// LS Electric XG5000 project: 루시드 Test
// PLC NewPLC
// module base 0 slot 0: 입출력 모듈:XBM-DN32H (DC 24V입력/TR 출력, 32점)

PROGRAM NewProgram (task: 스캔 프로그램)

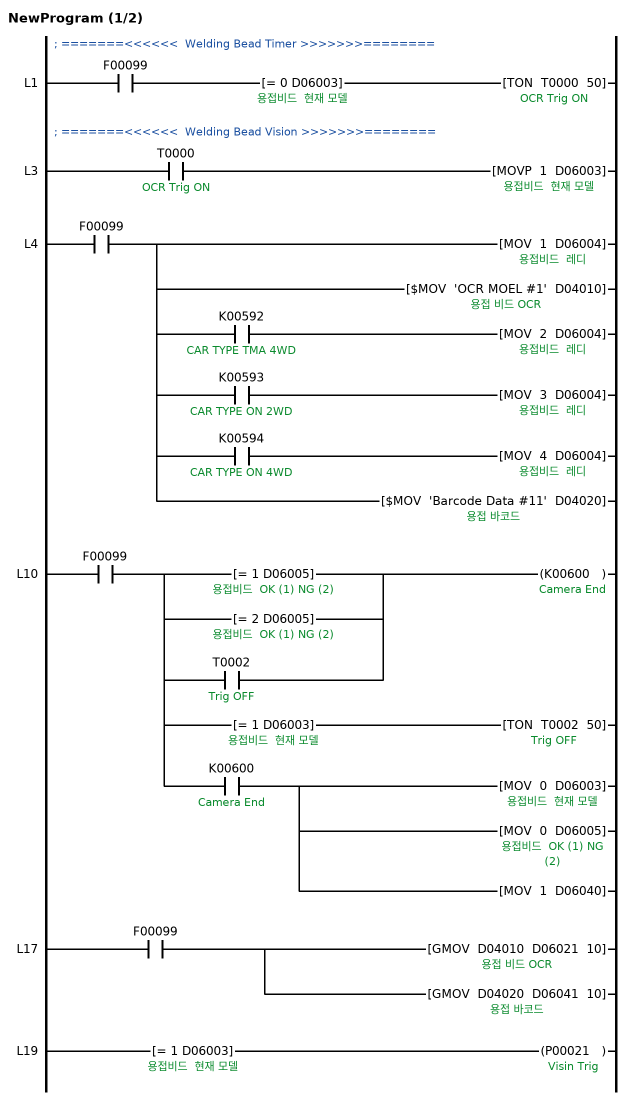
// =======<<<<<<  Welding Bead Timer >>>>>>>========
; L1
LOAD      F00099
AND=      0 D06003	// 용접비드  현재 모델
TON       T0000 50	// OCR Trig ON
// =======<<<<<<  Welding Bead Vision >>>>>>>========
; L3
LOAD      T0000	// OCR Trig ON
MOVP      1 D06003	// 용접비드  현재 모델
; L4
LOAD      F00099
MOV       1 D06004	// 용접비드  레디 
$MOV      'OCR MOEL #1' D04010	// 용접 비드 OCR
MPUSH
AND       K00592	// CAR TYPE TMA 4WD
MOV       2 D06004	// 용접비드  레디 
MLOAD
AND       K00593	// CAR TYPE ON 2WD
MOV       3 D06004	// 용접비드  레디 
MLOAD
AND       K00594	// CAR TYPE ON 4WD
MOV       4 D06004	// 용접비드  레디 
MPOP
$MOV      'Barcode Data #11' D04020	// 용접 바코드
; L10
LOAD      F00099
MPUSH
LOAD=     1 D06005	// 용접비드  OK (1) NG (2)
OR=       2 D06005	// 용접비드  OK (1) NG (2)
OR        T0002	// Trig OFF
AND LOAD
OUT       K00600	// Camera End
MLOAD
AND=      1 D06003	// 용접비드  현재 모델
TON       T0002 50	// Trig OFF
MPOP
AND       K00600	// Camera End
MOV       0 D06003	// 용접비드  현재 모델
MOV       0 D06005	// 용접비드  OK (1) NG (2)
MOV       1 D06040
; L17
LOAD      F00099
GMOV      D04010 D06021 10	// 용접 비드 OCR
GMOV      D04020 D06041 10	// 용접 바코드
; L19
LOAD=     1 D06003	// 용접비드  현재 모델
OUT       P00021	// Visin Trig

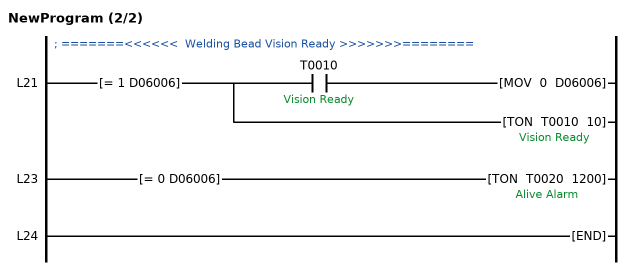
// =======<<<<<<  Welding Bead Vision Ready >>>>>>>========
; L21
LOAD=     1 D06006
MPUSH
AND       T0010	// Vision Ready
MOV       0 D06006
MPOP
TON       T0010 10	// Vision Ready
; L23
LOAD=     0 D06006
TON       T0020 1200	// Alive Alarm
; L24
END

VARIABLES AND COMMENTS (devices not used above)
D06000	WORD	용접비드  촬영 (1: 전송 0:PC)
D06001	WORD	용접비드  OCR 전송
D06002	WORD	용접비드  바코드 전송
K00591	BIT	CAR TYPE TMA 2WD
T0001	BIT/WORD	Welding Bead Trig ON
P00020	BIT	OCR Trig
D06010	WORD	용접비드  OCR DATA #1
D06011	WORD	용접비드  OCR DATA #2
D06012	WORD	용접비드  OCR DATA #3
D06013	WORD	용접비드  OCR DATA #4
D06020	WORD	용접비드  바코드 #1